FUNCTION_BLOCK ABSTRACT ZAppSequence EXTENDS ZApplication.Sequence IMPLEMENTS ZCore.ISequence

METHOD StepDecoded : ZCore.ZString
VAR_INPUT
  stepIndex : INT;
END_VAR
VAR_INST
  _stepIndexDecoded : ZAppStep;
END_VAR
_stepIndexDecoded := stepIndex;
StepDecoded := TO_STRING(_stepIndexDecoded);
END_METHOD

END_FUNCTION_BLOCK

(* stored: Version 1.1.0.1
   POU ZAppSequence: Id {6875e96e-d2c2-4f25-9fb1-f6e8ed96fde8}, SpecialFunc None
   Method StepDecoded: Id {841d67e8-d280-4eec-a0a9-6d4d12816c69} *)
